PROGRAM MAIN
VAR
		my_counter : INT := 0;
END_VAR

my_counter := my_counter + my_counter + my_counter + 1;

END_PROGRAM

(* stored: Version 1.1.0.1, ProductVersion 3.1.4024.12
   POU MAIN: Id {c8cb04b9-63d8-4b8b-8792-b29c5e8af7b2}, SpecialFunc None *)
